SUBAPPLICATION Uebung_034a2 (* Numeric Value Input auf PWM Ausgang *)
  (* Standard: 61499-2 *)
  (* Version 1.0, 2023-10-23, franz *)
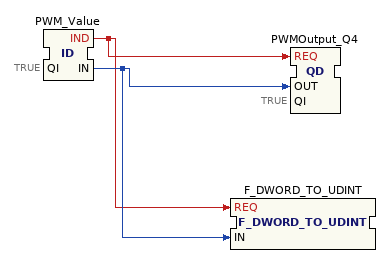
  (* ACHTUNG !! IND erscheint erst, wenn man die Numeric Value mit OK Bestätigt. nicht bei Button Druck. *)
  FBS
    F_DWORD_TO_UDINT : F_DWORD_TO_UDINT;
    PWMOutput_Q4 : QD(QI := TRUE);
    PWM_Value : ID(QI := TRUE);
  END_FBS
  EVENT_CONNECTIONS
    PWM_Value.IND TO PWMOutput_Q4.REQ;
    PWM_Value.IND TO F_DWORD_TO_UDINT.REQ;
  END_CONNECTIONS
  DATA_CONNECTIONS
    PWM_Value.IN TO F_DWORD_TO_UDINT.IN;
    PWM_Value.IN TO PWMOutput_Q4.OUT;
  END_CONNECTIONS
END_SUBAPPLICATION
